(* PLC project Basic LD rung, react-plc-diagram PLCopen XML test fixtures 0.1.0 *)
(* stored: creationDateTime 2026-08-12T00:00:00Z, modificationDateTime 2026-08-12T00:00:00Z *)

PROGRAM BasicRung
  VAR
    Start : BOOL;
    Motor : BOOL;
  END_VAR

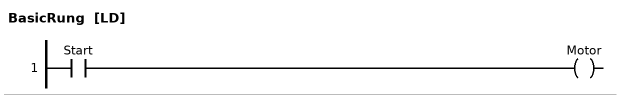
(* LD diagram, written out as Structured Text *)
Motor := Start;
END_PROGRAM
